(* Logix 5000 project; controller PLC2_Project_10_PumpProtection Emulate 5570 rev 20.11; software revision 20.00 *)
// Project 10: Pump protection

TASK MainTask (continuous, watchdog 500 ms) : MainProgram

MODULES
   Local : Emulate 5570 (ICP 1, rev 20.11)
END_MODULES

ADD_ON_INSTRUCTION NSCP   (* revision 1.0 *)
// Nicks Scale With Parameters
VAR_INPUT
   InputMax : REAL; {required}
   InputMin : REAL; {required}
   ScaledMaxOut : REAL; {required}
   ScaledMinOut : REAL; {required}
   Input : REAL; {required}
END_VAR
VAR_OUTPUT
   ScaledOutput : REAL; {access Read Only, required}
END_VAR
VAR
   Rate : REAL; {access None}
END_VAR

ROUTINE Logic   (* structured text *)
   // My scale with parameters
   IF (EnableIn) THEN
   	Rate := (ScaledMaxOut - ScaledMinOut) / (InputMax - InputMin);
   	ScaledOutput := (Input - InputMin) * Rate + ScaledMinOut;
   END_IF;
END_ROUTINE
END_ADD_ON_INSTRUCTION

PROGRAM MainProgram   (* main routine _00_Main *)
VAR
   _IN_A_PressureSensor : DINT; {access Read Only}
   _IN_FlowSwitchLL : BOOL; {access Read Only}
   _IN_PB_AlarmReset : BOOL; {access Read Only}
   _IN_PB_AlarmSilence : BOOL; {access Read Only}
   _IN_PB_HOA_Auto : BOOL; {access Read Only}
   _IN_PB_HOA_Hand : BOOL; {access Read Only}
   _IN_PB_HOA_Off : BOOL; {access Read Only}
   _ONS_FlowLLNotify : BOOL; {access Read Only}
   _ONS_HOA_Auto : BOOL; {access Read Only}
   _ONS_HOA_Off : BOOL; {access Read Only}
   _ONS_HoaLastState : BOOL; {access Read Only}
   _ONS_NotHandMode : BOOL; {access Read Only}
   _ONS_PresHHNotify : BOOL; {access Read Only}
   _OUT_FlowFaultIndicator : BOOL; {access Read Only}
   _OUT_PressureFaultIndicator : BOOL; {access Read Only}
   _OUT_PumpEn : BOOL; {access Read Only}
   Alarm_Notify_Silence : BOOL; {access Read Only}
   Alarm_Reset : BOOL; {access Read Only}
   CycleMode : DINT; {access Read Only}   // 0 = Off/Waiting 1 = Pump En 30s 2 = Pump off 10s
   HOA_LastState : DINT; {access Read Only}
   HOA_Mode : DINT; {access Read Only}   // 0 = Off 1 = Hand 2 = Auto
   HOA_PB_Auto : BOOL; {access Read Only}
   HOA_PB_Hand : BOOL; {access Read Only}
   HOA_PB_Off : BOOL; {access Read Only}
   Pump_Alarm_Flow_LL : BOOL; {access Read Only}
   Pump_Alarm_Press_HH : BOOL; {access Read Only}
   Pump_AlarmNotify_FlowFault : BOOL; {access Read Only}
   Pump_AlarmNotify_PressureFault : BOOL; {access Read Only}
   Pump_Cycle_EnTimer : TIMER := (PRE := 10000); {access Read Only}
   Pump_Cycle_OffTimer : TIMER := (PRE := 5000); {access Read Only}
   Pump_En : BOOL; {access Read Only}
   Pump_Flow_LL_AlarmTimer : TIMER := (PRE := 5000); {access Read Only}
   Pump_FlowSwitch_HH : BOOL; {access Read Only}
   Pump_Pressure : REAL; {access Read Only}   // 0 - 55 PSI Sensor at outgoing pump
   Pump_Pressure_HH_AlarmTimer : TIMER := (PRE := 5000); {access Read Only}
   Pump_Pressure_NSCP : NSCP; {access Read Only}
END_VAR

ROUTINE _00_Main   (* ladder *)
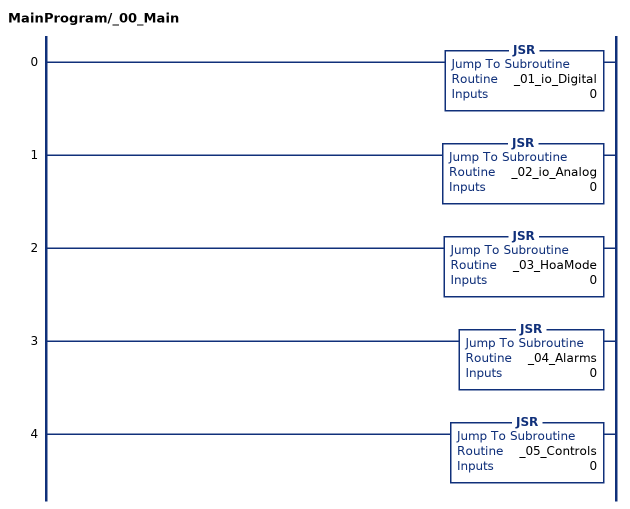
   0: JSR(_01_io_Digital,0);
   1: JSR(_02_io_Analog,0);
   2: JSR(_03_HoaMode,0);
   3: JSR(_04_Alarms,0);
   4: JSR(_05_Controls,0);
END_ROUTINE

ROUTINE _01_io_Digital   (* ladder *)
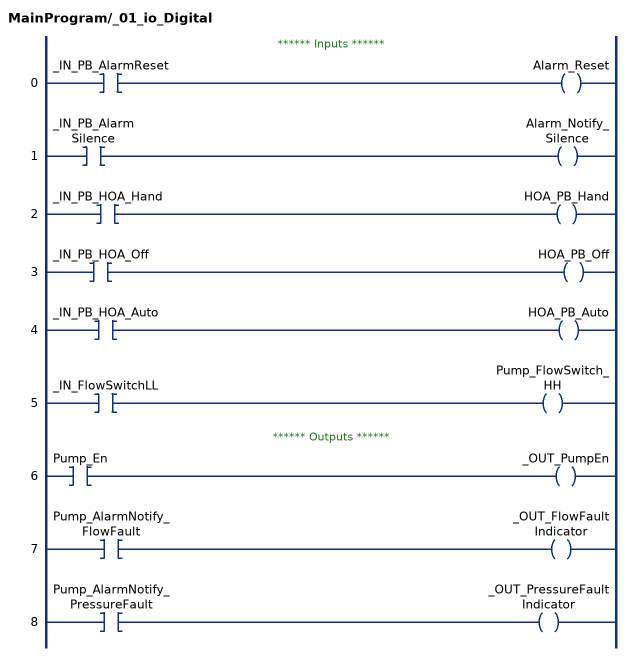
   // ****** Inputs ******
   0: XIC(_IN_PB_AlarmReset)OTE(Alarm_Reset);
   1: XIC(_IN_PB_AlarmSilence)OTE(Alarm_Notify_Silence);
   2: XIC(_IN_PB_HOA_Hand)OTE(HOA_PB_Hand);
   3: XIC(_IN_PB_HOA_Off)OTE(HOA_PB_Off);
   4: XIC(_IN_PB_HOA_Auto)OTE(HOA_PB_Auto);
   5: XIC(_IN_FlowSwitchLL)OTE(Pump_FlowSwitch_HH);
   // ****** Outputs ******
   6: XIC(Pump_En)OTE(_OUT_PumpEn);
   7: XIC(Pump_AlarmNotify_FlowFault)OTE(_OUT_FlowFaultIndicator);
   8: XIC(Pump_AlarmNotify_PressureFault)OTE(_OUT_PressureFaultIndicator);
END_ROUTINE

ROUTINE _02_io_Analog   (* ladder *)
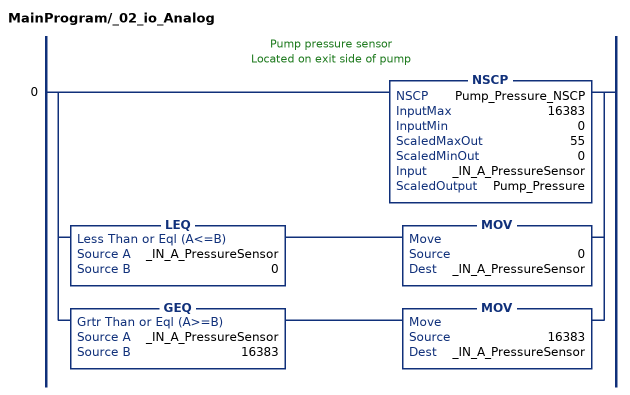
   // Pump pressure sensor
   // Located on exit side of pump
   0: [NSCP(Pump_Pressure_NSCP,16383,0,55,0,_IN_A_PressureSensor,Pump_Pressure) ,LEQ(_IN_A_PressureSensor,0) MOV(0,_IN_A_PressureSensor) ,GEQ(_IN_A_PressureSensor,16383) MOV(16383,_IN_A_PressureSensor) ];
END_ROUTINE

ROUTINE _03_HoaMode   (* ladder *)
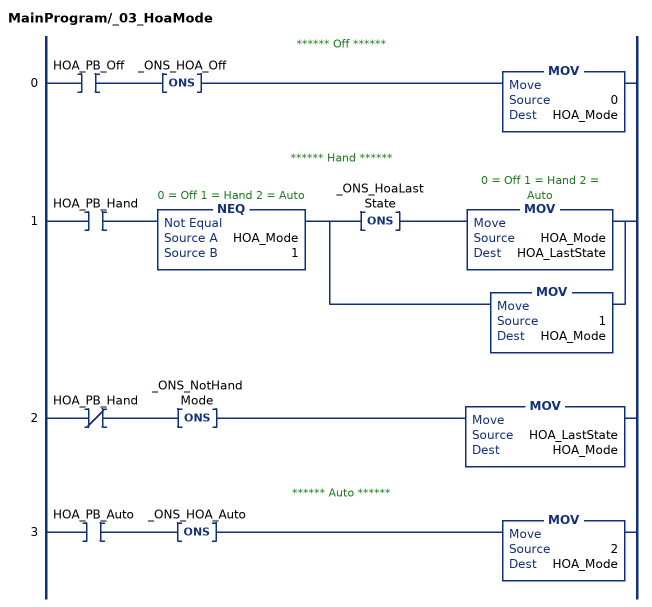
   // ****** Off ******
   0: XIC(HOA_PB_Off)ONS(_ONS_HOA_Off)MOV(0,HOA_Mode);
   // ****** Hand ******
   1: XIC(HOA_PB_Hand)NEQ(HOA_Mode,1)[ONS(_ONS_HoaLastState) MOV(HOA_Mode,HOA_LastState) ,MOV(1,HOA_Mode) ];
   2: XIO(HOA_PB_Hand)ONS(_ONS_NotHandMode)MOV(HOA_LastState,HOA_Mode);
   // ****** Auto ******
   3: XIC(HOA_PB_Auto)ONS(_ONS_HOA_Auto)MOV(2,HOA_Mode);
END_ROUTINE

ROUTINE _04_Alarms   (* ladder *)
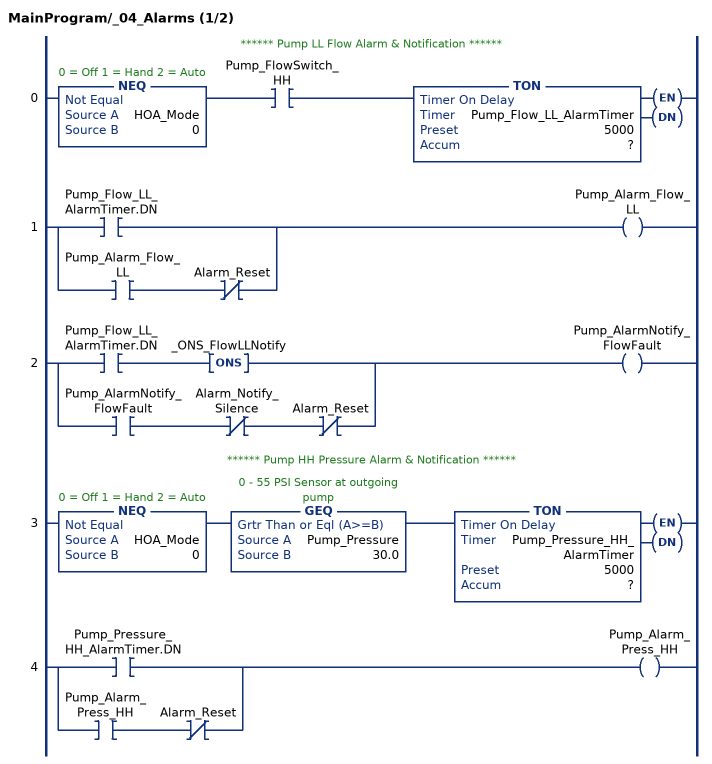
   // ****** Pump LL Flow Alarm & Notification ******
   0: NEQ(HOA_Mode,0)XIC(Pump_FlowSwitch_HH)TON(Pump_Flow_LL_AlarmTimer,?,?);
   1: [XIC(Pump_Flow_LL_AlarmTimer.DN) ,XIC(Pump_Alarm_Flow_LL) XIO(Alarm_Reset) ]OTE(Pump_Alarm_Flow_LL);
   2: [XIC(Pump_Flow_LL_AlarmTimer.DN) ONS(_ONS_FlowLLNotify) ,XIC(Pump_AlarmNotify_FlowFault) XIO(Alarm_Notify_Silence) XIO(Alarm_Reset) ]OTE(Pump_AlarmNotify_FlowFault);
   // ****** Pump HH Pressure Alarm & Notification ******
   3: NEQ(HOA_Mode,0)GEQ(Pump_Pressure,30.0)TON(Pump_Pressure_HH_AlarmTimer,?,?);
   4: [XIC(Pump_Pressure_HH_AlarmTimer.DN) ,XIC(Pump_Alarm_Press_HH) XIO(Alarm_Reset) ]OTE(Pump_Alarm_Press_HH);
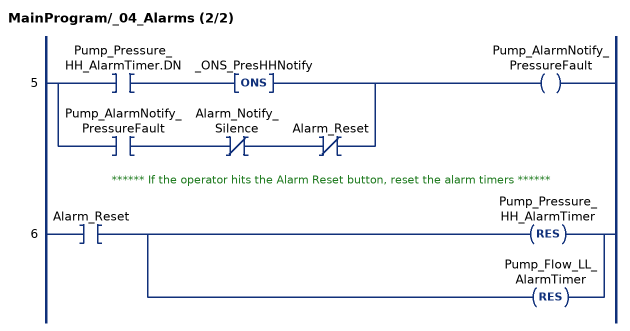
   5: [XIC(Pump_Pressure_HH_AlarmTimer.DN) ONS(_ONS_PresHHNotify) ,XIC(Pump_AlarmNotify_PressureFault) XIO(Alarm_Notify_Silence) XIO(Alarm_Reset) ]OTE(Pump_AlarmNotify_PressureFault);
   // ****** If the operator hits the Alarm Reset button, reset the alarm timers ******
   6: XIC(Alarm_Reset)[RES(Pump_Pressure_HH_AlarmTimer) ,RES(Pump_Flow_LL_AlarmTimer) ];
END_ROUTINE

ROUTINE _05_Controls   (* ladder *)
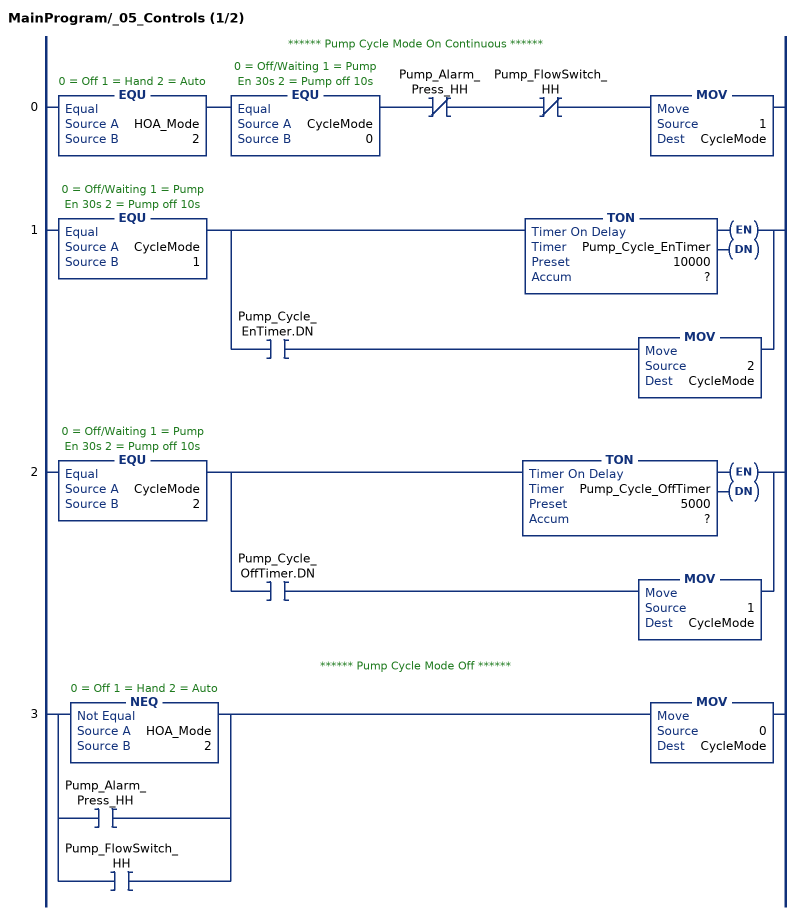
   // ****** Pump Cycle Mode On Continuous ******
   0: EQU(HOA_Mode,2)EQU(CycleMode,0)XIO(Pump_Alarm_Press_HH)XIO(Pump_FlowSwitch_HH)MOV(1,CycleMode);
   1: EQU(CycleMode,1)[TON(Pump_Cycle_EnTimer,?,?) ,XIC(Pump_Cycle_EnTimer.DN) MOV(2,CycleMode) ];
   2: EQU(CycleMode,2)[TON(Pump_Cycle_OffTimer,?,?) ,XIC(Pump_Cycle_OffTimer.DN) MOV(1,CycleMode) ];
   // ****** Pump Cycle Mode Off ******
   3: [NEQ(HOA_Mode,2) ,XIC(Pump_Alarm_Press_HH) ,XIC(Pump_FlowSwitch_HH) ]MOV(0,CycleMode);
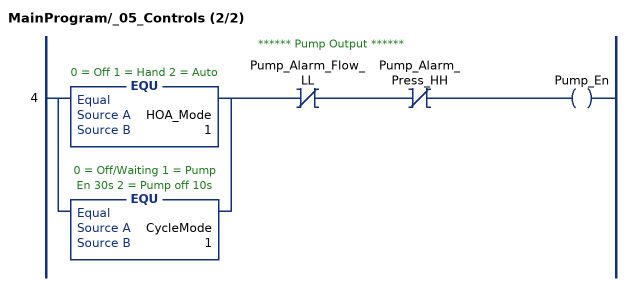
   // ****** Pump Output ******
   4: [EQU(HOA_Mode,1) ,EQU(CycleMode,1) ]XIO(Pump_Alarm_Flow_LL)XIO(Pump_Alarm_Press_HH)OTE(Pump_En);
END_ROUTINE
END_PROGRAM
